FUNCTION alg_a_pusher1 : BOOL
VAR_INPUT
	state: STATE;
END_VAR

alg_a_pusher1 := FALSE;

END_FUNCTION

(* stored: Version 1.1.0.1, ProductVersion 3.1.4022.18
   POU alg_a_pusher1: Id {9f34d037-e0b0-4ce4-ad4e-c7dc7fdea8ff}, SpecialFunc None *)
